PROGRAM MAIN
VAR
CheckXas:CheckStatusVanHetSysteem;
END_VAR

CheckXas();

END_PROGRAM

(* stored: Version 1.1.0.1, ProductVersion 3.1.4024.12
   POU MAIN: Id {2e858929-44f3-4765-9260-56aa5ca04b48}, SpecialFunc None *)
